FUNCTION_BLOCK FB_Ampel
VAR_INPUT
	Ampel_Rot				: BOOL;
	Ampel_Orange			: BOOL;
	Ampel_Gruen				: BOOL;
	Ampel_Blau				: BOOL;
	Ampel_Buzz				: BOOL;
END_VAR
VAR_OUTPUT
	{attribute 'OPC.UA.DA' := '1'} Steuerung				: ST_Ampel_Steuerung;			
	{attribute 'OPC.UA.DA' := '1'} Zustand					: ST_Ampel_Zustand;				
END_VAR
VAR
	OUT_Stellung_Rot			AT %Q* : BOOL;
	OUT_Stellung_Orange			AT %Q* : BOOL;
	OUT_Stellung_Gruen			AT %Q* : BOOL;
	OUT_Stellung_Blau			AT %Q* : BOOL;
	OUT_Stellung_Buzz			AT %Q* : BOOL;

	SchreibeDaten		: FB_Ampel_Out;
END_VAR

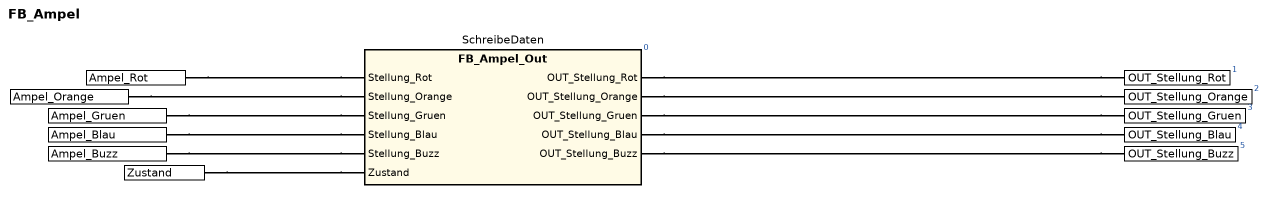
SchreibeDaten(
    Stellung_Rot := Ampel_Rot,
    Stellung_Orange := Ampel_Orange,
    Stellung_Gruen := Ampel_Gruen,
    Stellung_Blau := Ampel_Blau,
    Stellung_Buzz := Ampel_Buzz,
    Zustand := Zustand); // FB_Ampel_Out
OUT_Stellung_Rot := SchreibeDaten.OUT_Stellung_Rot;
OUT_Stellung_Orange := SchreibeDaten.OUT_Stellung_Orange;
OUT_Stellung_Gruen := SchreibeDaten.OUT_Stellung_Gruen;
OUT_Stellung_Blau := SchreibeDaten.OUT_Stellung_Blau;
OUT_Stellung_Buzz := SchreibeDaten.OUT_Stellung_Buzz;

END_FUNCTION_BLOCK

(* stored: Version 1.1.0.1, ProductVersion 3.1.4024.9
   POU FB_Ampel: Id {9a2845ff-3025-419e-bd87-9a2b7b41424d}, SpecialFunc None *)
